FUNCTION LDT_TO_STRING : STRING(24)
VAR_INPUT
	uliTime	:	ULINT; 	//Time [ms]
END_VAR
VAR
	dtTime			:	DATE_AND_TIME;
	uliMillisecond	:	ULINT;
	sTime			:	STRING(24);
END_VAR

IF uliTime = 0 THEN
	LDT_TO_STRING := '-';
	RETURN;
END_IF
dtTime := ULINT_TO_DT(uliTime/1000);
uliMillisecond := uliTime - DT_TO_ULINT(dtTime);
sTime := DT_TO_STRING(dtTime);
sTime := DELETE(sTime,3,1);
sTime := CONCAT(sTime,'.');
if uliMillisecond = 0 then
	sTime := CONCAT(sTime,'000');
ELSIF uliMillisecond < 100 THEN
	sTime := CONCAT(sTime,'0');
	sTime := CONCAT(sTime,ULINT_TO_STRING(uliMillisecond));
ELSE
	sTime := CONCAT(sTime,ULINT_TO_STRING(uliMillisecond));	
END_IF
LDT_TO_STRING := sTime;

END_FUNCTION

(* stored: Version 1.1.0.1, ProductVersion 3.1.4024.9
   POU LDT_TO_STRING: Id {7cac4314-166c-4fbd-b81f-6ed1690347a4}, SpecialFunc None *)
